FUNCTION_BLOCK L3_FaultyMHDLR (* Basic Function Block Type *)
  (* Standard: 61499-2 *)
  (* Version 0.0, 2014-10-06, EQUEROL, UJI *)
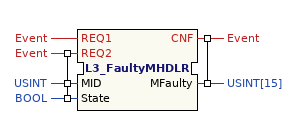
  EVENT_INPUT
    REQ1; (* Request from core to update faulty machines vector *)
    REQ2 WITH MID, State; (* Indicates a change in the state of a machine *)
  END_EVENT
  EVENT_OUTPUT
    CNF WITH MFaulty; (* Execution Confirmation *)
  END_EVENT
  VAR_INPUT
    MID : USINT; (* Faulty machine identifier *)
    State : BOOL; (* Machine state *)
  END_VAR
  VAR_OUTPUT
    MFaulty : ARRAY [0..14] OF USINT; (* Faulty machines vector *)
  END_VAR
  VAR
    FaultyMachines : ARRAY [0..14] OF USINT := [0,0,0,0,0,0,0,0,0,0,0,0,0,0,0]; (* Internal Variable *)
    i : USINT; (* loop variable *)
  END_VAR
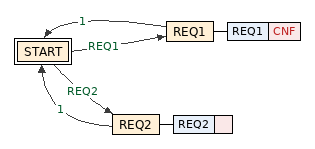
  EC_STATES
    START; (* Initial State *)
    REQ1 : REQ1 -> CNF; (* Normal execution *)
    REQ2 : REQ2;
  END_STATES
  EC_TRANSITIONS
    START TO REQ1 := REQ1;
    REQ1 TO START := 1;
    START TO REQ2 := REQ2;
    REQ2 TO START := 1;
  END_TRANSITIONS
  ALGORITHM REQ1 IN ST: (* Update core machine state vector *)
(*This algo send to the core the changes in the machine state since last call*)
FOR i := 0 TO 14 DO
		MFaulty[i] := FaultyMachines[i];
		FaultyMachines[i] := 0;
END_FOR;
  END_ALGORITHM
  ALGORITHM REQ2 IN ST: (* Handles the arrival of changes in machine status *)
IF State = true THEN
	(*Machine repaired*)
	FaultyMachines[MID] := 2;
ELSE
	(*Machine breakdown*)
	FaultyMachines[MID] := 1;
END_IF;
  END_ALGORITHM
END_FUNCTION_BLOCK
